FUNCTION_BLOCK FB_SimMotion
VAR_INPUT
	iAdvanceReq:BOOL;
	iReturnReq:BOOL;
	iClear:BOOL;
	
END_VAR

VAR_OUTPUT
	qAdvanced:BOOL;
	qReturned:BOOL;
END_VAR
VAR
	timAdvanceDelay: TON;
	timReturnDelay: TON;
END_VAR

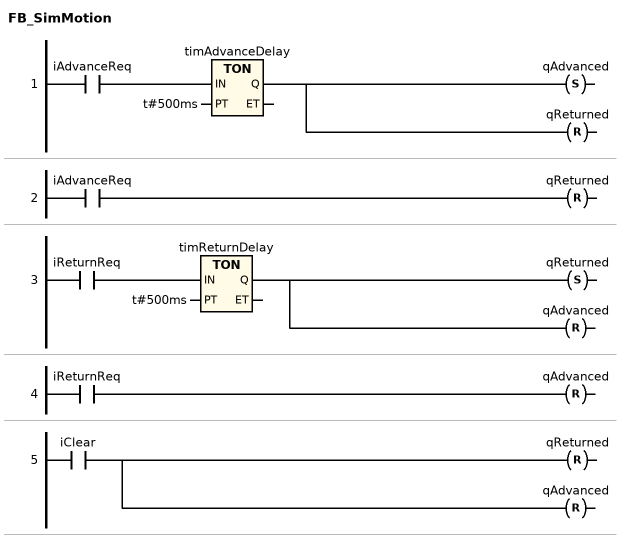
// NETWORK 1
timAdvanceDelay(IN := iAdvanceReq, PT := t#500ms); // TON
qAdvanced S= timAdvanceDelay.Q;
qReturned R= timAdvanceDelay.Q;

// NETWORK 2
qReturned R= iAdvanceReq;

// NETWORK 3
timReturnDelay(IN := iReturnReq, PT := t#500ms); // TON
qReturned S= timReturnDelay.Q;
qAdvanced R= timReturnDelay.Q;

// NETWORK 4
qAdvanced R= iReturnReq;

// NETWORK 5
qReturned R= iClear;
qAdvanced R= iClear;

END_FUNCTION_BLOCK

(* stored: Version 1.1.0.1, ProductVersion 3.1.4024.11
   POU FB_SimMotion: Id {2747f1a0-b71c-03b4-2bbe-7ed49864bb3c}, SpecialFunc None *)
